// TIA Portal V16 export
// export: Created 2023-08-28T09:37:48.141585Z, ExportSetting WithDefaults, DisplayName Totally Integrated Automation Portal, DisplayVersion V16 Update 6, DisplayName TIA Portal Version Control Interface, DisplayVersion V16 Update 2, DisplayName TIA Portal Openness, DisplayVersion V16 Update 6, DisplayName STEP 7 Professional, DisplayVersion V16 Update 6, DisplayName STEP 7 Safety, DisplayVersion V16, DisplayName WinCC Advanced, DisplayVersion V16 Update 6
DATA_BLOCK "dbSterowanie dołaczaniem dodatkocych_FB1"   // DB3
AUTHOR : RTecmer
FAMILY : Ster
VERSION : 0.1
// stored: AutoNumber true, DBAccessibleFromOPCUA true, InstanceOfName 06_M_Control of switching on an additional pump, InstanceOfType FB
"06_M_Control of switching on an additional pump"
   // VAR_INPUT
   //    daneMV { ExternalAccessible := 'False'; ExternalVisible := 'False'; ExternalWritable := 'False'} : Real;
   //    trybPracyPID { ExternalAccessible := 'False'; ExternalVisible := 'False'; ExternalWritable := 'False'} : Int;
   //    IsMode_Aut { ExternalAccessible := 'False'; ExternalVisible := 'False'; ExternalWritable := 'False'} : Bool;
   //    IsReady_F1 { ExternalAccessible := 'False'; ExternalVisible := 'False'; ExternalWritable := 'False'} : Bool;
   //    InputWarning_H_PID { ExternalAccessible := 'False'; ExternalVisible := 'False'; ExternalWritable := 'False'} : Bool;
   //    InputWarning_L_PID { ExternalAccessible := 'False'; ExternalVisible := 'False'; ExternalWritable := 'False'} : Bool;
   //    Timer_K1 { ExternalAccessible := 'False'; ExternalVisible := 'False'; ExternalWritable := 'False'} : Time;
   //    Timer_K2 { ExternalAccessible := 'False'; ExternalVisible := 'False'; ExternalWritable := 'False'} : Time;
   //    Timer_K3 { ExternalAccessible := 'False'; ExternalVisible := 'False'; ExternalWritable := 'False'} : Time;
   //    Timer_OFF_K1 { ExternalAccessible := 'False'; ExternalVisible := 'False'; ExternalWritable := 'False'} : Time;
   //    Timer_OFF_K2 { ExternalAccessible := 'False'; ExternalVisible := 'False'; ExternalWritable := 'False'} : Time;
   //    Timer_OFF_K3 { ExternalAccessible := 'False'; ExternalVisible := 'False'; ExternalWritable := 'False'} : Time;
   //    Time_50Hz { ExternalAccessible := 'False'; ExternalVisible := 'False'; ExternalWritable := 'False'} : Time;
   //    IsAuto_P1 : Bool;
   //    IsAuto_P2 : Bool;
   //    IsAuto_P3 : Bool;
   //    IsAuto_P4 : Bool;
   //    Mem_K1 : Bool;
   //    IsIncrease : Bool;
   //    CureentQ1 : Word;
   //    IsRunInverterMA : Bool;
   //    IsRunInverterMB : Bool;
   //    IsRunInverterMC : Bool;
   //    IsRunInverterMD : Bool;
   //    IsReady_MA : Bool;
   //    IsReady_MB : Bool;
   //    IsReady_MC : Bool;
   //    IsReady_MD : Bool;
   //    Rst_Motor2_Alarm : Bool;
   //    Rst_Motor3_Alarm : Bool;
   //    Rst_Motor4_Alarm : Bool;
   //    correction_reset_K1 : Real;
   //    correction_reset_K2 : Real;
   // END_VAR
   // VAR_IN_OUT
   //    Set_K1 { ExternalWritable := 'False'} : Bool;
   //    Set_K2 { ExternalWritable := 'False'} : Bool;
   //    Set_K3 : Bool;
   //    Set_K4 { ExternalWritable := 'False'} : Bool;
   // END_VAR
   // VAR
   //    Temp_bar_OFF { ExternalAccessible := 'False'; ExternalVisible := 'False'; ExternalWritable := 'False'} : Real;
   //    reset_Value_K1 { ExternalAccessible := 'False'; ExternalVisible := 'False'; ExternalWritable := 'False'} : Real;
   //    reset_Value_K2 { ExternalAccessible := 'False'; ExternalVisible := 'False'; ExternalWritable := 'False'} : Real;
   //    reset_value_K3 { ExternalAccessible := 'False'; ExternalVisible := 'False'; ExternalWritable := 'False'} : Real;
   //    table_index { ExternalAccessible := 'False'; ExternalVisible := 'False'; ExternalWritable := 'False'} : Int;
   //    WarningHigbar { ExternalAccessible := 'False'; ExternalVisible := 'False'; ExternalWritable := 'False'} : Real;
   //    isAvailable { ExternalAccessible := 'False'; ExternalVisible := 'False'; ExternalWritable := 'False'} : Bool;
   //    temp_reset_value_K3 { ExternalAccessible := 'False'; ExternalVisible := 'False'; ExternalWritable := 'False'} : Real;
   //    is_correctio_bar { ExternalAccessible := 'False'; ExternalVisible := 'False'; ExternalWritable := 'False'} : Bool;
   // END_VAR
BEGIN
END_DATA_BLOCK
